ABB RobotStudio station: RS1_11_2.rsstnx

Station RS1 (saved by RobotStudio 25.5.11605.0)
Controller IRB140_6_81
  mechanical unit ROB_1: IRB140_6_81_C_03, 6 joints, base frame (0, 0, 0) mm
Layout (positions relative to the parent item):
  - IRB140_6_81_C_03 [mechanism, from %ABB.RobotStudio.Models.IRB140%\IRB140_6_81_C_G_03.rslib] at (0, 0, 0) mm; joint values [0, 0.076, 0.0347, 0, 1.4601, 0] (rad or m)
  - UISpenholder [mechanism, from Components\UISpenholder (1).rslib] at (475, 0, 604) mm, rotated rx 180 ry 0 rz 180 deg
  - table_and_fixture_140 [part, from Training Objects\propeller_table.rslib] at (300, 225, 0) mm, rotated rx 0 ry 0 rz -90 deg
Attachment: UISpenholder is attached to IRB140_6_81_C_03 / Link6
Attachment: wobjTable is attached to table_and_fixture_140
Collision set CollisionSet_1: UISpenholder against table_and_fixture_140, near miss 0 m
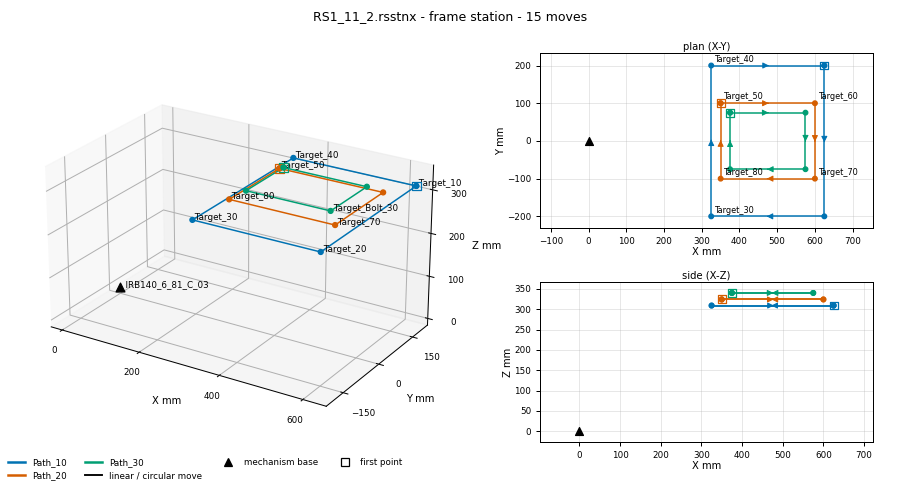
[picture p0: tool path of RS1_11_2.rsstnx in frame station, 15 of 15 moves have a stored position in this frame; points joined in program order, loops and branches not executed]
Targets, tools, work objects and paths stored in the station, written as RAPID:
! task T_ROB1
MODULE Module1
  PERS tooldata UISpenholder:=[TRUE,[[0,0,110],[1,0,0,0]],[1,[0,0,1],[1,0,0,0],0,0,0]];
  TASK PERS wobjdata wobjTable:=[FALSE,TRUE,"",[[325,200,309],[0.707106781,0,0,-0.707106781]],[[0,0,0],[1,0,0,0]]];
  CONST robtarget Target_10:=[[0,300,0],[0,-0.707106781,0.707106781,0],[0,0,0,0],[9E+09,9E+09,9E+09,9E+09,9E+09,9E+09]];
  CONST robtarget Target_20:=[[400,300,0],[0,-0.707106781,0.707106781,0],[-1,0,-1,0],[9E+09,9E+09,9E+09,9E+09,9E+09,9E+09]];
  CONST robtarget Target_30:=[[400,0,0],[0,-0.707106781,0.707106781,0],[-1,0,-1,0],[9E+09,9E+09,9E+09,9E+09,9E+09,9E+09]];
  CONST robtarget Target_40:=[[0,0,0],[0,-0.707106781,0.707106781,0],[0,0,0,0],[9E+09,9E+09,9E+09,9E+09,9E+09,9E+09]];
  CONST robtarget Target_50:=[[100,25,15],[0,-0.707106781,0.707106781,0],[0,0,-2,0],[9E+09,9E+09,9E+09,9E+09,9E+09,9E+09]];
  CONST robtarget Target_60:=[[100,275,15],[0,-0.707106781,0.707106781,0],[0,0,-2,0],[9E+09,9E+09,9E+09,9E+09,9E+09,9E+09]];
  CONST robtarget Target_70:=[[300,275,15],[0,-0.707106781,0.707106781,0],[-1,0,1,0],[9E+09,9E+09,9E+09,9E+09,9E+09,9E+09]];
  CONST robtarget Target_80:=[[300,25,15],[0,-0.707106781,0.707106781,0],[0,0,0,0],[9E+09,9E+09,9E+09,9E+09,9E+09,9E+09]];
  CONST robtarget Target_Bolt_10:=[[125,50,31],[0,1,0,0],[0,0,0,0],[9E+09,9E+09,9E+09,9E+09,9E+09,9E+09]];
  CONST robtarget Target_Bolt_20:=[[125,250,31],[0,1,0,0],[0,0,-1,0],[9E+09,9E+09,9E+09,9E+09,9E+09,9E+09]];
  CONST robtarget Target_Bolt_30:=[[275,250,31],[0,1,0,0],[-1,0,-2,0],[9E+09,9E+09,9E+09,9E+09,9E+09,9E+09]];
  CONST robtarget Target_Bolt_40:=[[275,50,31],[0,1,0,0],[-1,0,-2,0],[9E+09,9E+09,9E+09,9E+09,9E+09,9E+09]];
  CONST robtarget Target_ShaftAbove_10:=[[200,150,164],[0,1,0,0],[0,0,0,0],[9E+09,9E+09,9E+09,9E+09,9E+09,9E+09]];
  PROC Path_10()
    MoveL Target_10,v1000,z5,UISpenholder\WObj:=wobjTable;
    MoveL Target_20,v1000,z5,UISpenholder\WObj:=wobjTable;
    MoveL Target_30,v1000,z5,UISpenholder\WObj:=wobjTable;
    MoveL Target_40,v1000,z5,UISpenholder\WObj:=wobjTable;
    MoveL Target_10,v1000,z5,UISpenholder\WObj:=wobjTable;
  ENDPROC
  PROC main()
    Path_10;
  ENDPROC
  PROC Path_20()
    MoveL Target_50,v1000,z5,UISpenholder\WObj:=wobjTable;
    MoveL Target_60,v1000,z5,UISpenholder\WObj:=wobjTable;
    MoveL Target_70,v1000,z5,UISpenholder\WObj:=wobjTable;
    MoveL Target_80,v1000,z5,UISpenholder\WObj:=wobjTable;
    MoveL Target_50,v1000,z5,UISpenholder\WObj:=wobjTable;
  ENDPROC
  PROC Path_30()
    MoveL Target_Bolt_10,v1000,z100,UISpenholder\WObj:=wobjTable;
    MoveL Target_Bolt_20,v1000,z100,UISpenholder\WObj:=wobjTable;
    MoveL Target_Bolt_30,v1000,z100,UISpenholder\WObj:=wobjTable;
    MoveL Target_Bolt_40,v1000,z100,UISpenholder\WObj:=wobjTable;
    MoveL Target_Bolt_10,v1000,z100,UISpenholder\WObj:=wobjTable;
  ENDPROC
ENDMODULE

